{attribute 'qualified_only'}
{attribute 'strict'}
TYPE INTERNAL _EntityState :
(
	Unregistered,
	Registered,
	Completed
);
END_TYPE

(* stored: Version 1.1.0.1
   DUT _EntityState: Id {74c03052-379c-4bb4-b9b6-d250c4ffb73e} *)
